FUNCTION_BLOCK ABSTRACT FBA_TrifectaDrive EXTENDS FBA_Drive
VAR
	outerLimit AT %I* : BOOL;
END_VAR
(*
this abstract FB adds a rear limit sensor to FBA_Drive
*)

{attribute 'monitoring':='call'}
PROPERTY AtOuterLimit : BOOL
GET
AtOuterLimit := outerLimit <> limitSensorDefaultState;
END_GET
END_PROPERTY

END_FUNCTION_BLOCK

(* stored: Version 1.1.0.1, ProductVersion 3.1.4024.11
   POU FBA_TrifectaDrive: Id {585dcf41-d2f4-4504-9bc2-9bb00fb240d7}, SpecialFunc None
   Property AtOuterLimit: Id {881e2a21-3a15-4aaa-8087-01fda7b3148d}
   Get Get: Id {236a32da-b6d3-42b7-9bea-2b43ef51ea91} *)
